# B&R Automation Studio project lab1_kvbo_08_21
Automation Studio 4.5.2.102

## Configuration Config1

### Task classes (Cpu.sw)
```
Cyclic#2:
  Program <- Program.prg
  lab1 <- lab1.prg [disabled]
Binaries: udbdef, TCData, ashwd, User, asfw, arconfig, sysconf, Role, ashwac, iomap
Libraries: MotorCont
```

### Hardware
```
4PP065_0571_P74 : 4PP065.0571-P74 v1.1.2.0
  Connector IF5:
    ActivateDevice = 1
  ConfigurationID = lab1_kvbo_08_21_Config1
  Simulation = 1
```

## Logical view

Binary libraries used (declarations not repeated): operator, runtime, astime, AsIecCon

### Package Logical/Libraries - Global libraries

### Library Logical/Libraries/MotorCont (ANSIC)

#### MotorCont.fun - Exported functions and function blocks
```iecst
{REDUND_ERROR} FUNCTION_BLOCK FB_Integrator (*TODO: Add your comment here*) (*$GROUP=User,$CAT=User,$GROUPICON=User.png,$CATICON=User.png*)
	VAR_INPUT
		in : {REDUND_UNREPLICABLE} REAL; (*input integrator*)
	END_VAR
	VAR_OUTPUT
		out : {REDUND_UNREPLICABLE} REAL; (*output integrator*)
	END_VAR
	VAR
		dt : {REDUND_UNREPLICABLE} REAL; (*step in sec*)
		state : REAL;
	END_VAR
END_FUNCTION_BLOCK

{REDUND_ERROR} FUNCTION_BLOCK FB_Motor (*TODO: Add your comment here*) (*$GROUP=User,$CAT=User,$GROUPICON=User.png,$CATICON=User.png*)
	VAR_INPUT
		u : REAL; (*input voltage [v]*)
	END_VAR
	VAR_OUTPUT
		w : {REDUND_UNREPLICABLE} REAL; (*frequency of revolving [rev/min]*)
		phi : {REDUND_UNREPLICABLE} REAL; (*position [rad]*)
	END_VAR
	VAR
		integrator : FB_Integrator; (*integrator*)
		Tm : REAL; (*el_mech const of time [sec]*)
		ke : REAL; (*EDS of motor [V*min/rev]*)
		dt : REAL; (*step of calculation [sec]*)
	END_VAR
END_FUNCTION_BLOCK

{REDUND_ERROR} FUNCTION_BLOCK FB_Regulator (*TODO: Add your comment here*) (*$GROUP=User,$CAT=User,$GROUPICON=User.png,$CATICON=User.png*)
	VAR_INPUT
		e : REAL; (*dissonance between input and real speed of motor revolving [rev/min]*)
	END_VAR
	VAR_OUTPUT
		u : {REDUND_UNREPLICABLE} REAL; (*voltage goes in motor [v]*)
	END_VAR
	VAR
		k_i : REAL; (*integral coef*)
		k_p : REAL; (*proprtional coef*)
		integrator : FB_Integrator; (*integrator*)
		iyOld : REAL; (*previous state*)
		max_abs_value : REAL; (*border of restriction block [v]*)
		dt : REAL; (*step of calculation*)
	END_VAR
END_FUNCTION_BLOCK
```

#### FB_Integrator.c
```c
#include <bur/plctypes.h>
#ifdef __cplusplus
	extern "C"
	{
#endif
	#include "MotorCont.h"
#ifdef __cplusplus
	};
#endif
/* TODO: Add your comment here */
void FB_Integrator(struct FB_Integrator* inst)
{
	/*TODO: Add your code here*/
	inst->dt=0.01;
	inst->out = inst->dt*inst->in + inst->state;
	inst->state = inst->out;
}
```

#### FB_Motor.c
```c
#include <bur/plctypes.h>
#ifdef __cplusplus
	extern "C"
	{
#endif
	#include "MotorCont.h"
#ifdef __cplusplus
	};
#endif
/* TODO: Add your comment here */
void FB_Motor(struct FB_Motor* inst)
{
	/*motor*/
	REAL buf1 = inst->u*(1/inst->ke) - inst->w;
	REAL buf2 = buf1/inst->Tm;

	inst->integrator.in = buf2;
	FB_Integrator(&inst->integrator);

	inst->w = inst->integrator.out;

	/*speed sensor*/
	inst->integrator.in = inst->w;
	FB_Integrator(&inst->integrator);

	inst->phi = inst->integrator.out;

}
```

#### FB_Regulator.c
```c
#include <bur/plctypes.h>
#ifdef __cplusplus
	extern "C"
	{
#endif
	#include "MotorCont.h"
#ifdef __cplusplus
	};
#endif
/* TODO: Add your comment here */
void FB_Regulator(struct FB_Regulator* inst)
{
	/*TODO: Add your code here*/
	REAL buf_up = inst->e*inst->k_p;
	REAL buf_down = inst->e*inst->k_i;
	if (buf_up > inst->max_abs_value || buf_up < -inst->max_abs_value)
	{
		if (buf_up > 0) buf_up = inst->max_abs_value;
		else buf_up = -inst->max_abs_value;
	}

	buf_down = buf_down+inst->iyOld;

	inst->integrator.in = buf_down;
	FB_Integrator(&inst->integrator);

	buf_down = inst->integrator.out;

	REAL buf = buf_up+buf_down;

	if (buf > inst->max_abs_value || buf < -inst->max_abs_value)
	{
		if (buf > 0) buf = inst->max_abs_value;
		else buf = -inst->max_abs_value;
		inst->u = buf;
	}
	else
	{
		inst->u = buf;
	}
	inst->iyOld = inst->u-buf;

}
```

### Program Logical/lab1 (ANSIC)

#### Variables.var
```iecst
VAR
	fb_motor : FB_Motor;
	integrator : FB_Integrator;
	fb_controller : FB_Regulator;
	enable : BOOL;
	speed : REAL;
	fb_motor2 : FB_Motor;
	counter : REAL;
	speed1 : REAL;
END_VAR
```

#### Cyclic.c
```c
#include <bur/plctypes.h>

#ifdef _DEFAULT_INCLUDES
	#include <AsDefault.h>
#endif

void _CYCLIC ProgramCyclic(void)
{
	if(enable == 1)
	{
		counter+=1;
		if (counter >= 500 && counter <= 1000) speed1 = 40;
		else speed1 = 5;
	}

	else speed1 = 0;
	fb_controller.e = speed1 - fb_motor.w;
	fb_motor2.u = speed1*fb_motor2.ke;
	fb_motor.u = fb_controller.u * fb_motor.ke;
	FB_Regulator(&fb_controller);
	FB_Motor(&fb_motor);
	FB_Motor(&fb_motor2);
}
```

#### Init.c
```c
#include <bur/plctypes.h>

#ifdef _DEFAULT_INCLUDES
	#include <AsDefault.h>
#endif

void _INIT ProgramInit(void)
{
	enable=1;
	counter=0;
	speed=0;
	fb_motor.dt=0.02;
	fb_motor.ke=5;
	fb_motor.Tm=0.05;
	fb_motor2.dt=0.02;
	fb_motor2.ke=5;
	fb_motor2.Tm=0.05;

	fb_controller.dt=0.02;
	fb_controller.k_p=0.0064;
	fb_controller.k_i=0.16;
	fb_controller.max_abs_value=24;
}
```

### Program Logical/Program (ANSIC)

#### Main.c
```c
#include <bur/plctypes.h>

#ifdef _DEFAULT_INCLUDES
	#include <AsDefault.h>
#endif

void _INIT ProgramInit(void)
{
	enable=1;
	counter=0;
	speed=0;
	fb_motor.dt=0.01;
	fb_motor.ke=43.98;
	fb_motor.Tm=0.173;
	fb_motor2.dt=0.01;
	fb_motor2.ke=43.98;
	fb_motor2.Tm=0.173;

	fb_controller.dt=0.02;
	fb_controller.k_p=3.804;
	fb_controller.k_i =21.99;
	fb_controller.max_abs_value=24;
}

void _CYCLIC ProgramCyclic(void)
{
	if(enable == 1)
	{
		counter+=1;
		if (counter >= 500 && counter <= 1000) speed1 = 40;
		else speed1 = 5;
	}

	else speed1 = 0;
	fb_controller.e = speed1 - fb_motor.w;
	fb_motor2.u = speed1*fb_motor2.ke;
	fb_motor.u = fb_controller.u * fb_motor.ke;
	FB_Regulator(&fb_controller);
	FB_Motor(&fb_motor);
	FB_Motor(&fb_motor2);
}

void _EXIT ProgramExit(void)
{

}
```

Listed in the project but not available here: Logical/Global.typ, Logical/Global.var, Logical/Libraries/MotorCont/Types.typ, Logical/Libraries/MotorCont/Constants.var
